FUNCTION_BLOCK MyBlink
VAR_INPUT
	tBlinkTime			: TON;
	bEnable				: BOOL;
	bBlinkHz			: BOOL;
	tTimeOn				: TIME := T#2S;
	tTimeOff 			: TIME := tTimeOn/2;
END_VAR
VAR_OUTPUT
	bBlink				: BOOL;
END_VAR
VAR
END_VAR

// SET Timer ON
tBlinkTime(IN:=NOT tBlinkTime.Q, PT:= tTimeON);

// Set Timer OFF
bBlinkHz := tBlinkTime.ET >= tTimeOff;

// OUTPUT
bBlink := bBlinkHz AND bEnable;

END_FUNCTION_BLOCK

(* stored: Version 1.1.0.1, ProductVersion 3.1.4024.12
   POU MyBlink: Id {f2b54b98-3b3b-4032-b38c-5cb30df8dd76}, SpecialFunc None *)
